// TIA Portal V15.1 export
// export: Created 2024-06-21T08:40:53.6250373Z, ExportSetting WithDefaults, DisplayName Totally Integrated Automation Portal, DisplayVersion V15.1 Update 5, DisplayName TIA Portal Openness, DisplayVersion V15.1 Update 5, DisplayName SINAMICS Startdrive Advanced, DisplayVersion V15.1, DisplayName G130, G150, S120, S150, SINAMICS MV, S210, DisplayVersion V15.1, DisplayName G110M, G120, G120C, G120D, G120P, DisplayVersion V15.1, DisplayName STEP 7 Professional, DisplayVersion V15.1 Update 5, DisplayName STEP 7 Safety, DisplayVersion V15.1, DisplayName WinCC Professional, DisplayVersion V15.1 Update 5, DisplayName SIMATIC Visualization Architect, DisplayVersion V15.1
FUNCTION "LSimpleIAnim" : Void   // FC1009, FBD
TITLE = LSimpleIAnim
{ S7_Optimized_Access := 'FALSE' }
AUTHOR : VCC
FAMILY : Control
NAME : SIAnim
VERSION : 1.0
// ================================================================================
// Handles the conversion from bits to one Word for simple icon animation. 
// ================================================================================
// stored: AutoNumber false, IsIECCheckEnabled false, SetENOAutomatically False, UDAEnableTagReadback false
   VAR_INPUT
      I_SetPos : Bool;   // Set position
      I_ResetPos : Bool;   // Reset position
      I_Active : Bool;   // Active
      I_Invisible : Bool;   // Invisible
      I_OutOfUse : Bool;   // Object out of use
      I_AlarmA : Bool;   // AlarmA
      I_AlarmB : Bool;   // AlarmB
      I_AlarmC : Bool;   // AlarmC
      I_AlarmD : Bool;   // AlarmD
      I_ManualMode : Bool;   // Manual mode
      I_FncSelInHMI : Bool;   // Manual selection from HMI
   END_VAR
   VAR_OUTPUT
      H_IAnim : Word;   // Icon animation Word
   END_VAR
BEGIN

REGION Network 1: **** 8 - Outputs **** Set position
   // Set position
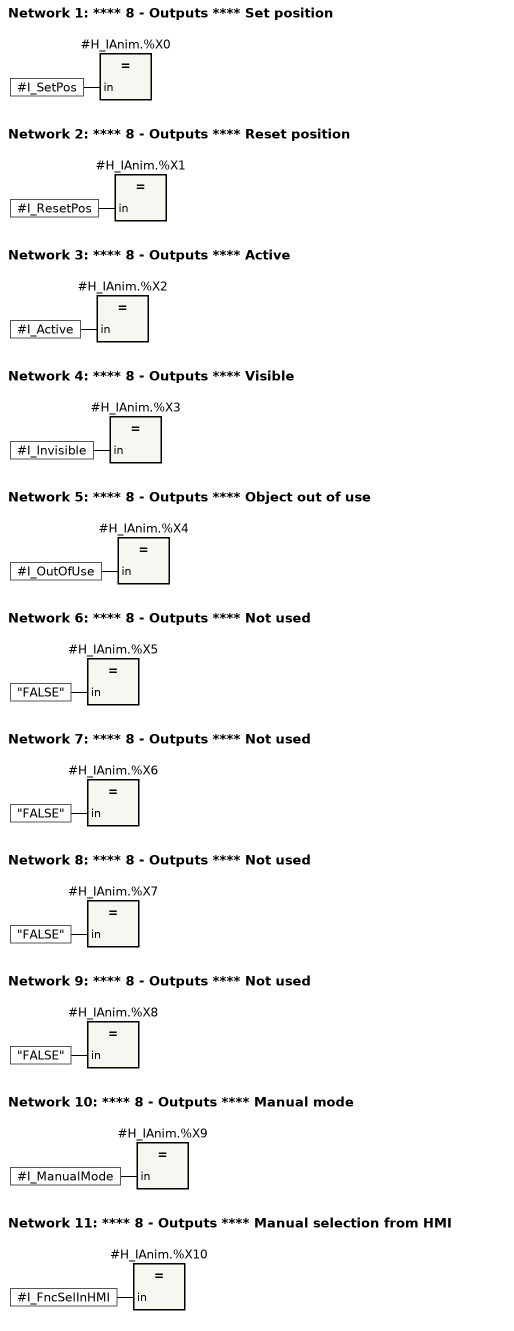
   #H_IAnim.%X0 := #I_SetPos;
END_REGION

REGION Network 2: **** 8 - Outputs **** Reset position
   // Reset position
   #H_IAnim.%X1 := #I_ResetPos;
END_REGION

REGION Network 3: **** 8 - Outputs **** Active
   // Active
   #H_IAnim.%X2 := #I_Active;
END_REGION

REGION Network 4: **** 8 - Outputs **** Visible
   // Visible
   #H_IAnim.%X3 := #I_Invisible;
END_REGION

REGION Network 5: **** 8 - Outputs **** Object out of use
   // Object out of use
   #H_IAnim.%X4 := #I_OutOfUse;
END_REGION

REGION Network 6: **** 8 - Outputs **** Not used
   // Not used
   #H_IAnim.%X5 := "FALSE";
END_REGION

REGION Network 7: **** 8 - Outputs **** Not used
   // Not used
   #H_IAnim.%X6 := "FALSE";
END_REGION

REGION Network 8: **** 8 - Outputs **** Not used
   // Not used
   #H_IAnim.%X7 := "FALSE";
END_REGION

REGION Network 9: **** 8 - Outputs **** Not used
   // Not used
   #H_IAnim.%X8 := "FALSE";
END_REGION

REGION Network 10: **** 8 - Outputs **** Manual mode
   // Manual mode
   #H_IAnim.%X9 := #I_ManualMode;
END_REGION

REGION Network 11: **** 8 - Outputs **** Manual selection from HMI
   // Manual selection from HMI
   #H_IAnim.%X10 := #I_FncSelInHMI;
END_REGION

REGION Network 12: **** 8 - Outputs **** Not used
   // Not used
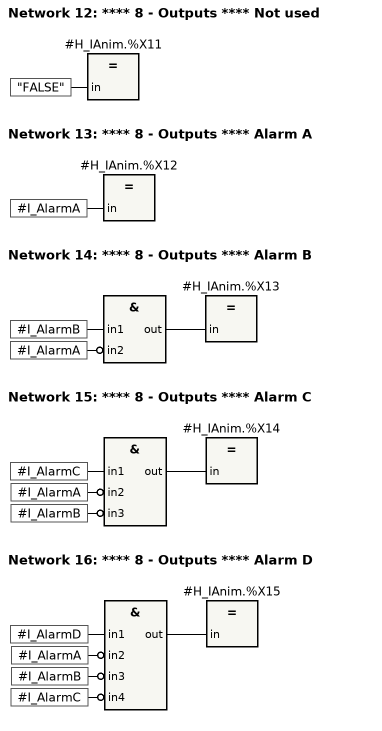
   #H_IAnim.%X11 := "FALSE";
END_REGION

REGION Network 13: **** 8 - Outputs **** Alarm A
   // Alarm A
   #H_IAnim.%X12 := #I_AlarmA;
END_REGION

REGION Network 14: **** 8 - Outputs **** Alarm B
   // Alarm B
   #H_IAnim.%X13 := #I_AlarmB AND NOT #I_AlarmA;
END_REGION

REGION Network 15: **** 8 - Outputs **** Alarm C
   // Alarm C
   #H_IAnim.%X14 := #I_AlarmC AND NOT #I_AlarmA AND NOT #I_AlarmB;
END_REGION

REGION Network 16: **** 8 - Outputs **** Alarm D
   // Alarm D
   #H_IAnim.%X15 := #I_AlarmD AND NOT #I_AlarmA AND NOT #I_AlarmB AND NOT #I_AlarmC;
END_REGION
END_FUNCTION
